// TIA Portal V20 export
FUNCTION_BLOCK "CompValEqOr"   // FB55, LAD
TITLE = COMP_VAL_==_OR_FB / COMP_VAL_==_OR
AUTHOR : SICAR
FAMILY : Miscellaneous
VERSION : 1.0
// Der Baustein vergleicht die Werte der Eingänge in1...in8 mit dem Wert des Eingangs „compareValue“ und verodert diese Vergleiche. Ist mindestens einer der Werte von in1...in8 gleich mit „compareValue“, so wird der Wert von „compareValue“ in den Output „value“ geschrieben. Andernfalls wird er mit dem Wert 0 beschrieben.  
// Anwendungsfall Beispiel: Damit kann ein "Summensignal" gebildet werden, z.B. für Produktionsdaten "Grenzwerte", womit ein Button animiert werden kann (Button "ProdData", "Grenzwerte").  
// 
// **Beispielaufruf**  
// Abbildung in Kontaktplan (KOP), ohne Parameterbeschaltung.  
// 
// **Aufrufschnittstelle**  
// Der Baustein wird im zyklischen Programm aufgerufen. In den Startup-Projekten ist der Baustein aufgerufen, für die Bildung eines Sammelsignals für die Grenzwerte der Produktionsdaten. Damit werden die Buttons  [ProdData]
// Compare the values of the inputs with the value of th input _compareValue_ generating a collective OR signal from these comparisons.
// stored: IsIECCheckEnabled true, MemoryReserve 100, SetENOAutomatically true
   VAR_INPUT
      compareValue { ExternalAccessible := 'False'; ExternalVisible := 'False'; ExternalWritable := 'False'} : UInt;   // Vergleichs Wert / Compare value
      val1 { ExternalAccessible := 'False'; ExternalVisible := 'False'; ExternalWritable := 'False'} : UInt;   // Wert 1 / value 1
      val2 { ExternalAccessible := 'False'; ExternalVisible := 'False'; ExternalWritable := 'False'} : UInt;   // Wert 2 / value 2
      val3 { ExternalAccessible := 'False'; ExternalVisible := 'False'; ExternalWritable := 'False'} : UInt;   // Wert 3 / value 3
      val4 { ExternalAccessible := 'False'; ExternalVisible := 'False'; ExternalWritable := 'False'} : UInt;   // Wert 4 / value 4
      val5 { ExternalAccessible := 'False'; ExternalVisible := 'False'; ExternalWritable := 'False'} : UInt;   // Wert 5 / value 5
      val6 { ExternalAccessible := 'False'; ExternalVisible := 'False'; ExternalWritable := 'False'} : UInt;   // Wert 6 / value 6
      val7 { ExternalAccessible := 'False'; ExternalVisible := 'False'; ExternalWritable := 'False'} : UInt;   // Wert 7 / value 7
      val8 { ExternalAccessible := 'False'; ExternalVisible := 'False'; ExternalWritable := 'False'} : UInt;   // Wert 8 / value 8
   END_VAR
   VAR_OUTPUT
      value { ExternalAccessible := 'False'; ExternalVisible := 'False'; ExternalWritable := 'False'} : UInt;   // Ergebnis Wert / Result value
   END_VAR
   VAR_TEMP
      tempDummy : Bool;   // Dummy
   END_VAR
BEGIN

REGION Network 1: Aufruf: Initialisierung SPS / ChangeLog
   // SIEMENS AG / (c)Copyright 2023
   // ------------------------------------------------------------------------------
   // Title:            CompValEqOr (FB55)
   // Comment/Function: Compare the values of the inputs with the value of th input compareValue generating a collective OR signal from these comparisons.
   // Library/Family:   Automation Framework
   // Author:           Siemens Digital Industry
   // Tested with:      ---
   // Engineering:      TIA Portal V19
   // Restrictions:     -
   // Requirements:     ---
   // ------------------------------------------------------------------------------
   // Change log table:
   // Version  | Date       | Expert in charge       | Changes applied
   // ---------|------------|------------------------|------------------------------
   // 01.00.00 | 11.12.2023 | Siemens Industry Online Support
   //                         First released version
END_REGION

REGION Network 2: Beschreibung / Description
   // The block compares the values of the inputs _in1 ... in8_ with the value of the input _compareValue_ and generates a collective OR signal from these comparisons. If at least one of the values of in1 ... in8 is equal with _compareValue_, the value of _compareValue_ is written to output “value”.  
   // Otherwise, “value” is written with the value 0.  
   // Use Case example: With this, a "summary signal" can be formed, e.g. for production data "Limit Values", with which a button can be animated (Button "ProdData", "LimitValues"). 
   // 
   // **Block call example**  
   // 
   // The call is shown as “Ladder Diagram” (LAD), without parameters.  
   // 
   // **Calling interface**  
   // 
   // The block is called in the cyclic program. In the startup projects, the block is called to generate a collective signal for the limit values of the production data. The buttons [ProdData] and [LimitValues] are animated in color, depending on the value range of the limit values.
   // 
   // **Operation mode Automatic / Manual**  
   // 
   // The block is independent of operation modes. Therefor it is not assigned to any operation mode area.
END_REGION

REGION Network 3: VALUE = 0 schreiben / set VALUE = 0
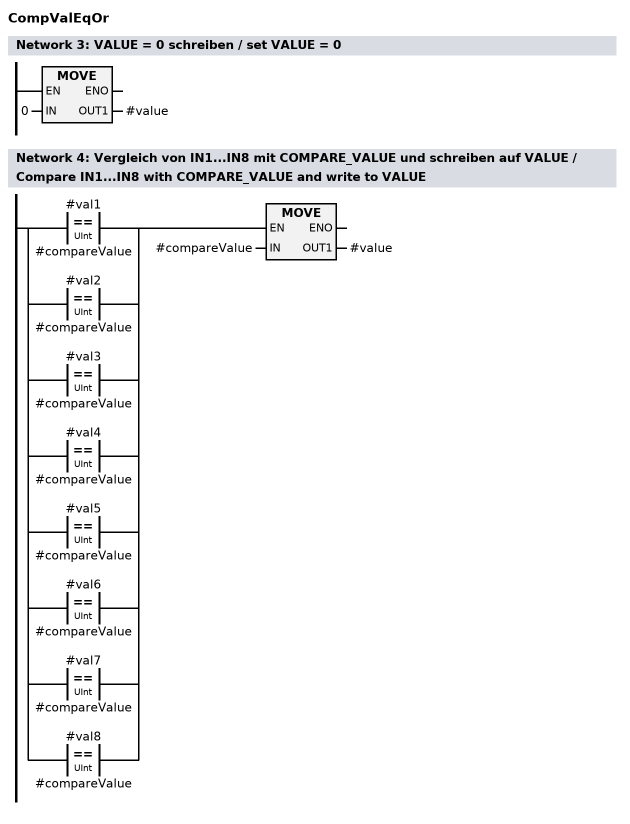
   RUNG wire#powerrail
      Move(in := 0, out1 => #value)
   END_RUNG
   // the same network as SCL:
   #value := 0;
END_REGION

REGION Network 4: Vergleich von IN1...IN8 mit COMPARE_VALUE und schreiben auf VALUE / Compare IN1...IN8 with COMPARE_VALUE and write to VALUE
   RUNG wire#powerrail
      { S7_Templates := "SrcType := UInt" } EQ_Contact(in1 := #val1, in2 := #compareValue)
      wire#w1
      Move(in := #compareValue, out1 => #value)
   END_RUNG
   RUNG wire#powerrail
      { S7_Templates := "SrcType := UInt" } EQ_Contact(in1 := #val2, in2 := #compareValue)
   END_RUNG wire#w1
   RUNG wire#powerrail
      { S7_Templates := "SrcType := UInt" } EQ_Contact(in1 := #val3, in2 := #compareValue)
   END_RUNG wire#w1
   RUNG wire#powerrail
      { S7_Templates := "SrcType := UInt" } EQ_Contact(in1 := #val4, in2 := #compareValue)
   END_RUNG wire#w1
   RUNG wire#powerrail
      { S7_Templates := "SrcType := UInt" } EQ_Contact(in1 := #val5, in2 := #compareValue)
   END_RUNG wire#w1
   RUNG wire#powerrail
      { S7_Templates := "SrcType := UInt" } EQ_Contact(in1 := #val6, in2 := #compareValue)
   END_RUNG wire#w1
   RUNG wire#powerrail
      { S7_Templates := "SrcType := UInt" } EQ_Contact(in1 := #val7, in2 := #compareValue)
   END_RUNG wire#w1
   RUNG wire#powerrail
      { S7_Templates := "SrcType := UInt" } EQ_Contact(in1 := #val8, in2 := #compareValue)
   END_RUNG wire#w1
   // the same network as SCL:
   IF (#val1 = #compareValue) OR (#val2 = #compareValue) OR (#val3 = #compareValue) OR (#val4 = #compareValue) OR (#val5 = #compareValue) OR (#val6 = #compareValue) OR (#val7 = #compareValue) OR (#val8 = #compareValue) THEN
       #value := #compareValue;
   END_IF;
END_REGION
END_FUNCTION_BLOCK
